(* PLC project PLC, Beckhoff Automation GmbH TwinCAT PLC Control 3.5.13.20 *)
(* stored: creationDateTime 2021-05-23T16:49:04.8482187, modificationDateTime 2021-05-23T16:49:04.9231855 *)

FUNCTION_BLOCK FB_Lamp
VAR_INPUT
END_VAR
VAR_OUTPUT
END_VAR

Fuck you my freind
Dont be sad

Again

VAR
END_VAR

            
          
END_FUNCTION_BLOCK
